PROGRAM MAIN
VAR
END_VAR

END_PROGRAM

(* stored: Version 1.1.0.1
   POU MAIN: Id {78bbdc00-e1e0-4c35-8ef1-9e7853b56e4e} *)
